Yaskawa INFORM job: N_R2_D50&56B(110_90,180).JBI

/JOB
//NAME N_R2_D50&56B(110_90,180)
//POS
///NPOS 227,227,227,10,0,0
///TOOL 0
///POSTYPE PULSE
///PULSE
C00000=22584,-91029,-87060,-7956,68824,61093
C00001=22584,-91029,-87060,-7956,68824,61093
C00002=2000,-113621,-91819,0,89172,0
C00003=-100725,-66745,-65547,-5330,101330,-31581
C00004=-137248,-37413,-60851,-11800,108062,-53976
C00005=-138411,-7940,-28391,-15115,116133,-60489
C00006=-180680,14026,-7685,-7917,112728,-80060
C00007=-186794,17026,42,-8794,108924,-82022
C00008=-187502,17265,3652,-8795,106773,-82119
C00009=-187502,17467,5395,-8744,105818,-82049
C00010=-182675,14939,3487,-14937,105773,-89393
C00011=-183307,13395,2083,-15043,105726,-89619
C00012=-186125,21667,9753,-10883,108766,-81970
C00013=-185415,19514,7722,-10739,109003,-81731
C00014=-186125,21667,9753,-10883,108766,-81970
C00015=-184476,23080,5547,-10788,112245,-81685
C00016=-135191,-11971,-32648,-15419,118418,-54869
C00017=-100725,-66745,-65547,-5330,101330,-31581
C00018=-68653,-71707,-73837,-24748,96021,-85891
C00019=-66615,-76041,-75906,-24722,95756,-75393
C00020=-80537,-30124,-13141,-12214,96831,-80465
C00021=-81172,-32496,-11329,-12285,94454,-80447
C00022=-81272,-33574,-9619,-12271,92868,-80323
C00023=-81272,-32874,-8019,-12261,92258,-80262
C00024=-81272,-33629,-9742,-12273,92916,-80327
C00025=-78377,-29561,-6671,-11651,93530,-79403
C00026=-82930,-25221,-2257,-8748,94612,-75231
C00027=-82159,-27675,-3939,-8560,94470,-74962
C00028=-82863,-25445,-2412,-8734,94601,-75208
C00029=-74565,-33759,-7503,-14334,89858,-83488
C00030=-75264,-34516,-7988,-14469,89651,-83703
C00031=-74565,-33759,-7503,-14334,89858,-83488
C00032=-74565,-35408,-11222,-14349,91256,-83650
C00033=-81291,-32137,-11094,-12310,94476,-80493
C00034=-172905,8912,9805,-17685,104206,-63243
C00035=-172925,6267,11032,-17511,102181,-62948
C00036=-173095,5120,12140,-17457,100932,-62826
C00037=-173095,5593,13541,-17414,100341,-62739
C00038=-172934,5281,11605,-17449,101360,-62831
C00039=-170941,3628,12252,-21342,95501,-69033
C00040=-171356,2541,11657,-21403,95212,-69131
C00041=-171898,950,10316,-21496,95078,-69302
C00042=-171356,2541,11657,-21403,95212,-69131
C00043=-173384,-23451,-12356,-17546,80818,-68289
C00044=-172173,-25440,-14096,-17586,81125,-67902
C00045=-171398,-26573,-14883,-17615,81198,-67636
C00046=-172724,-25294,-15625,-17531,81978,-68221
C00047=-143557,-6163,-8686,-20929,99946,-63784
C00048=-120837,-67343,-61251,1664,69818,-16688
C00049=-136948,17886,1372,-8158,95353,34817
C00050=-143935,27041,16447,-8009,90123,32767
C00051=-145422,30777,27912,-7980,84886,32590
C00052=-145422,32553,33696,-8012,82265,32756
C00053=-145422,33252,35771,-8025,81357,32815
C00054=-143676,31208,33052,-10858,81373,33518
C00055=-142910,30429,32946,-13100,80369,33952
C00056=-145422,32553,33696,-8012,82265,32756
C00057=-145422,30263,26046,-7974,85762,32534
C00058=-138335,26720,10522,-8993,93928,34380
C00059=-116233,-46119,-51802,-8224,97287,41779
C00060=-133480,-42640,-39007,-8140,89511,36383
C00061=-136265,-42532,-35298,-8104,87026,35591
C00062=-136265,-41955,-33217,-8108,86050,35653
C00063=-136265,-41609,-32030,-8111,85502,35689
C00064=-130241,-43052,-32167,-14495,84771,37934
C00065=-129806,-42953,-31605,-15984,84419,38162
C00066=-136265,-41955,-33217,-8108,86050,35653
C00067=-135498,-43523,-38278,-8113,88415,35764
C00068=-120126,-55162,-39521,-8172,84809,41259
C00069=-122393,-53466,-34860,-8212,82600,40629
C00070=-123299,-52550,-32544,-8233,81563,40387
C00071=-123299,-52047,-31285,-8241,81052,40420
C00072=-119861,-52196,-31542,-11446,81584,41751
C00073=-120901,-52203,-31545,-11457,81438,41408
C00074=-117579,-52136,-31515,-13326,82016,42591
C00075=-116541,-52768,-33293,-13289,82934,42851
C00076=-108480,-53248,-51729,-13121,95064,44368
C00077=-47420,-68885,-70906,-7741,99292,48439
C00078=-36237,-160244,-135216,-7095,93010,52660
C00079=-129093,-142421,-132565,-35762,109729,50782
C00080=-71329,-121440,-129553,-32440,109242,60016
C00081=-82746,-156345,-133581,-29501,88252,49791
C00082=-87611,-164628,-132694,-29771,81242,44951
C00083=-87611,-163220,-131273,-29779,81110,44987
C00084=-87611,-164709,-132775,-29767,81250,44951
C00085=-71886,-183234,-128665,-42620,74703,46418
C00086=-74833,-184908,-128996,-42921,72831,45887
C00087=-69878,-185821,-129175,-42644,74882,47243
C00088=-74429,-130912,-118044,-34983,110777,51627
C00089=-96642,-141369,-123481,-29522,97914,46607
C00090=-102270,-141697,-124015,-27978,95731,45009
C00091=-102270,-141154,-122872,-27952,95353,45100
C00092=-102270,-141737,-124103,-27981,95760,45001
C00093=-104565,-143039,-124460,-28044,94592,44404
C00094=-102270,-141737,-124103,-27981,95760,45001
C00095=-98711,-140115,-125335,-27931,98364,45740
C00096=-98711,-140115,-125335,-27931,98364,45740
C00097=-98939,-140108,-124921,-27921,98063,45725
C00098=-98939,-139729,-123974,-27889,97719,45808
C00099=-98939,-140167,-125070,-27927,98118,45710
C00100=-100683,-141421,-125418,-27980,97156,45273
C00101=-98939,-140167,-125070,-27927,98118,45710
C00102=-111795,-107890,-115236,-21941,123165,45716
C00103=-111980,-110192,-116037,-21807,122478,45790
C00104=-111795,-107890,-115236,-21941,123165,45716
C00105=-109061,-111903,-121767,-16718,119614,47923
C00106=-93191,-166945,-131033,-25725,96374,76077
C00107=-115036,-47760,-82622,-24757,104770,42999
C00108=-116312,-48104,-84043,-24644,105068,42493
C00109=-102840,-160852,-129487,-27293,95258,72668
C00110=-102950,-160931,-129604,-27308,95250,72628
C00111=-100000,-171791,-131669,-28056,90664,64085
C00112=-78747,-196536,-131709,-34622,83016,61742
C00113=-97788,-192520,-135527,-30708,76481,51692
C00114=-106746,-100694,-110680,-30872,101018,41696
C00115=-100997,-102592,-114676,-31446,104330,42992
C00116=-89249,-129083,-123995,-34588,91950,50732
C00117=-86172,-104791,-113024,-36662,97722,40982
C00118=-89586,-99522,-109974,-36341,97001,39840
C00119=-94829,-122476,-117865,-35334,89182,40270
C00120=-102758,-167765,-129707,-32742,64394,36090
C00121=-107366,-177085,-128987,-33295,58194,36082
C00122=-96698,-184464,-133250,-35581,61450,39784
C00123=-94800,-127534,-127780,-31715,84055,33612
C00124=-43155,-112421,-122950,-31185,87534,31974
C00125=-47420,-68885,-70906,-7741,99292,48439
C00126=-126000,-95781,-98048,7022,72166,-3406
C00127=-136814,-5298,6863,-118,87716,-82610
C00128=-137691,-48827,-35284,-2434,91122,-80550
C00129=-137775,-50491,-32454,-2438,88526,-80529
C00130=-144669,-59546,-36087,2970,81467,-83087
C00131=-137513,-49032,-30101,-2417,87837,-80428
C00132=-137980,-52740,-33271,-2456,87865,-80585
C00133=-136492,-62619,-37659,3141,80547,-80344
C00134=-130424,-52556,-33615,-1804,88372,-78049
C00135=-130538,-50934,-36491,-1816,90972,-78124
C00136=-134151,-85638,-58323,-18397,79452,-80216
C00137=-138797,-96086,-58203,-18217,70057,-80507
C00138=-132420,-53344,-33745,-21935,100560,-82879
C00139=-132280,-50606,-30920,-21871,100287,-82777
C00140=-143411,-94723,-57726,-17890,69450,-82098
C00141=-139141,-75011,-51892,-19052,86769,-83193
C00142=-144749,-26995,-11930,-14691,82144,-88756
C00143=-145691,-31856,-11979,-19284,78923,34918
C00144=-151034,-18823,4704,-13824,76424,32875
C00145=-151885,-17656,8121,-14166,75214,33243
C00146=-146071,-19738,8912,-19797,72571,35827
C00147=-147152,-20027,7322,-19728,73103,35349
C00148=-154357,-26510,2050,-14259,74004,32525
C00149=-152793,-10987,14638,-15716,82099,47051
C00150=-151339,-11562,10959,-15494,84269,47273
C00151=-146019,7566,32377,-21507,91583,49077
C00152=-147957,4386,28538,-22011,91765,48359
C00153=-147481,5615,30408,-21882,91404,48596
C00154=-144848,5152,34234,-24760,87902,50723
C00155=-159832,9049,31418,-7877,90076,62571
C00156=-198300,39103,67536,-4454,97929,51257
C00157=-197104,34479,56425,-4037,102437,51493
C00158=-197536,32116,56558,-4191,101125,51391
C00159=-198300,39103,67536,-4454,97929,51257
C00160=-197104,34479,56425,-4037,102437,51493
C00161=-145435,-6461,7890,-19316,88952,36538
C00162=-146400,-15498,9010,-17111,65695,33326
C00163=-150585,-15374,10170,-12685,65372,31387
C00164=-152770,-11869,15298,-10806,64283,30498
C00165=-148493,-14593,14125,-17227,62697,33002
C00166=-147445,-14270,15768,-17483,62104,33493
C00167=-150113,-3203,22864,-12407,64063,31649
C00168=-146055,-7115,17417,-17271,64938,33574
C00169=-149725,-15230,11944,-14152,64155,31991
C00170=-151735,-12378,15582,-12402,63542,31128
C00171=-148493,-14593,14125,-17227,62697,33002
C00172=-147444,-14270,15768,-17483,62104,33493
C00173=-151630,-3672,21747,-10124,65019,30743
C00174=-146194,-7735,16967,-17259,64868,33530
C00175=-147475,-4629,18347,-12944,66340,32408
C00176=-148206,-3042,20742,-12396,65722,32150
C00177=-144993,-5030,19536,-17422,64931,33970
C00178=-144005,-4679,21199,-17649,64331,34434
C00179=-147636,2823,25478,-11954,66212,32247
C00180=-159106,-19550,13776,8815,42964,19188
C00181=-160396,-25842,8024,9506,43156,18510
C00182=-160846,-38877,-8267,9186,46491,18652
C00183=-135242,-58896,-27541,-11024,46290,31048
C00184=-131236,-19716,-18108,-13510,71297,30401
C00185=-125742,9237,-5161,-19148,95170,30807
C00186=-133778,21116,12925,-19165,88751,28983
C00187=-139002,23165,16841,-12610,84259,27929
C00188=-139735,27050,26410,-12647,80339,28070
C00189=-131333,83852,86286,-19552,77576,31698
C00190=-130664,85028,89109,-19628,76664,32087
C00191=-140830,29311,28641,-10243,76630,19823
C00192=-140822,20487,15972,-10139,79847,19560
C00193=-137774,20952,11850,-14015,91367,38445
C00194=-140043,21612,21108,-13993,85767,38286
C00195=-131775,32332,27698,-18854,90275,38112
C00196=-132558,32274,26377,-18889,90837,37745
C00197=-141222,18370,18010,-13785,88896,43800
C00198=-140309,22876,20563,-13758,89776,44021
C00199=-138169,21721,13740,-13740,93646,44339
C00200=-130805,23103,4773,-14711,103608,44771
C00201=-116663,7219,3956,-17874,89187,41824
C00202=-120401,-109250,-97359,-24840,84473,3177
C00203=-33343,-40457,-55475,-21499,103344,-25825
C00204=-34531,-11543,-34459,-29967,106739,-58335
C00205=-34985,-14005,-32389,-29565,104365,-57871
C00206=-36737,-22261,-38534,-25905,98770,-56845
C00207=-35068,-14396,-32319,-29531,104124,-57840
C00208=-34264,-15859,-32209,-29394,103680,-57406
C00209=-37785,-26292,-41386,-25839,98165,-57100
C00210=-51408,-66161,-65218,-24804,88768,-60125
C00211=-46082,-52942,-64392,-25322,95990,-59686
C00212=-125318,-85686,-83357,-10390,89531,-85584
C00213=-142430,-46200,-62658,-6629,112309,-68083
C00214=-144446,-28774,-42147,-7166,118928,-64884
C00215=-142051,-28438,-38322,-12128,116138,-65491
C00216=-141798,-26650,-39491,-12256,117780,-65577
C00217=-132867,-37192,-45733,-18528,111034,-75329
C00218=-139736,-34425,-43384,-12199,112330,-75757
C00219=-134344,-42414,-48468,-16185,107501,-83449
C00220=-134440,-49684,-52823,-18552,102078,-90264
C00221=-130876,-45857,-53153,-18423,104940,-89409
C00222=-105687,-60080,-69740,-12786,102006,-79760
C00223=-4529,-28570,-46683,-27101,115691,-48588
C00224=2000,-113621,-91819,0,89172,0
C00225=2000,-113621,-91819,0,89172,0
C00226=2000,-113621,-91819,0,89172,0
BC00000=166445,688033,903774
BC00001=166445,688033,903774
BC00002=87189,714591,1075229
BC00003=279836,716878,248946
BC00004=347085,767945,248946
BC00005=351734,778369,248946
BC00006=397217,806013,248946
BC00007=397217,806013,248946
BC00008=397217,806013,248946
BC00009=397217,806013,248946
BC00010=397217,806013,248946
BC00011=397217,806013,248946
BC00012=397217,806013,248946
BC00013=397217,806013,248946
BC00014=397217,806013,248946
BC00015=397217,806013,248946
BC00016=347085,767945,248946
BC00017=279836,716878,248946
BC00018=74259,715122,420956
BC00019=74259,803457,420956
BC00020=74259,803457,420956
BC00021=74259,803457,420956
BC00022=74259,803457,420956
BC00023=74259,803457,420956
BC00024=74259,803457,420956
BC00025=74259,803457,420956
BC00026=74259,803457,420956
BC00027=74259,803457,420956
BC00028=74259,803457,420956
BC00029=74259,803457,420956
BC00030=74259,803457,420956
BC00031=74259,803457,420956
BC00032=74259,803457,420956
BC00033=74259,803457,420956
BC00034=168853,805006,369390
BC00035=168853,805006,369390
BC00036=168853,805006,369390
BC00037=168853,805006,369390
BC00038=168853,805006,369390
BC00039=168853,805006,369390
BC00040=168853,805006,369390
BC00041=168853,805006,369390
BC00042=168853,805006,369390
BC00043=168853,805006,369390
BC00044=168853,805006,369390
BC00045=168853,805006,369390
BC00046=168853,805006,369390
BC00047=153069,815778,383312
BC00048=89909,820992,348340
BC00049=133900,839476,347452
BC00050=133900,839476,347452
BC00051=133900,839476,347452
BC00052=133900,839476,347452
BC00053=133900,839476,347452
BC00054=133900,839476,347452
BC00055=133900,839476,347452
BC00056=133900,839476,347452
BC00057=133900,839476,347452
BC00058=133900,839476,347452
BC00059=91689,839476,305907
BC00060=91689,839476,305907
BC00061=91689,839476,305907
BC00062=91689,839476,305907
BC00063=91689,839476,305907
BC00064=91689,839476,305907
BC00065=91689,839476,305907
BC00066=91689,839476,305907
BC00067=91689,839476,305907
BC00068=65725,786338,350532
BC00069=65725,786338,350532
BC00070=65725,786338,350532
BC00071=65725,786338,350532
BC00072=65725,786338,350532
BC00073=65725,786338,350532
BC00074=65725,786338,350532
BC00075=65725,786338,350532
BC00076=65725,786338,350532
BC00077=45615,718562,524343
BC00078=45615,718562,1072524
BC00079=367621,718562,1072524
BC00080=396988,986746,1072524
BC00081=396988,986746,1072524
BC00082=396988,986746,1072524
BC00083=396988,986746,1072524
BC00084=396988,986746,1072524
BC00085=396988,986746,1072524
BC00086=396988,986746,1072524
BC00087=396988,986746,1072524
BC00088=396988,986746,1072524
BC00089=396982,986676,1072526
BC00090=396988,986746,1072524
BC00091=396988,986746,1072524
BC00092=396988,986746,1072524
BC00093=396988,986746,1072524
BC00094=396988,986746,1072524
BC00095=396988,986746,1072524
BC00096=396988,943028,1072524
BC00097=392786,943028,1061989
BC00098=392786,943028,1061989
BC00099=392786,943028,1061989
BC00100=392786,943028,1061989
BC00101=392786,943028,1061989
BC00102=392824,960696,1061989
BC00103=392824,960696,1061989
BC00104=392824,960696,1061989
BC00105=392827,960650,1061995
BC00106=397481,962635,1061991
BC00107=398174,909238,1075175
BC00108=398174,909238,1075175
BC00109=397481,962635,1061991
BC00110=397481,962635,1061991
BC00111=397481,962635,1061991
BC00112=397481,962635,1061991
BC00113=397481,962635,1061991
BC00114=397481,962635,1061991
BC00115=397481,962635,1061991
BC00116=397481,962635,1061991
BC00117=397481,962635,1061991
BC00118=397481,962635,1061991
BC00119=397481,962635,1061991
BC00120=397481,962635,1061991
BC00121=397481,962635,1061991
BC00122=397481,962635,1061991
BC00123=397481,917581,1061991
BC00124=298896,713787,1061991
BC00125=45615,718562,524343
BC00126=94279,727282,315353
BC00127=135603,815672,503004
BC00128=127958,797752,374153
BC00129=127958,797752,374153
BC00130=127958,797752,374153
BC00131=127958,797752,374153
BC00132=127958,797752,374153
BC00133=127958,797752,374153
BC00134=127958,797752,374153
BC00135=127958,797752,374153
BC00136=104823,825619,320967
BC00137=104823,825619,320967
BC00138=104823,825619,320967
BC00139=104823,825619,320967
BC00140=104823,825619,320967
BC00141=104823,825619,320967
BC00142=130544,787227,441208
BC00143=131883,785229,447466
BC00144=131883,785229,447466
BC00145=131883,785229,447466
BC00146=131883,785229,447466
BC00147=131883,785229,447466
BC00148=131883,785229,447466
BC00149=131883,785229,447466
BC00150=131883,785229,447466
BC00151=131883,785229,447466
BC00152=131883,785229,447466
BC00153=131883,785229,447466
BC00154=131883,785229,447466
BC00155=131883,785229,447466
BC00156=178294,839754,448603
BC00157=178294,839754,448603
BC00158=178294,839754,448603
BC00159=178294,839754,448603
BC00160=178294,839754,448603
BC00161=133874,781474,455608
BC00162=135864,777719,463750
BC00163=135864,777719,463750
BC00164=135864,777719,463750
BC00165=135864,777719,463750
BC00166=135864,777719,463750
BC00167=135864,777719,463750
BC00168=135864,777719,463750
BC00169=135957,805967,463073
BC00170=135957,805967,463073
BC00171=135957,805967,463073
BC00172=135957,805967,463073
BC00173=135957,805967,463072
BC00174=135957,805967,463073
BC00175=132965,820164,450481
BC00176=132965,820164,450481
BC00177=132965,820164,450481
BC00178=132965,820164,450481
BC00179=132965,820164,450481
BC00180=132965,820164,450481
BC00181=132965,820164,450481
BC00182=132965,820164,450481
BC00183=132965,820164,450481
BC00184=129716,827479,399778
BC00185=124610,838973,320111
BC00186=124537,838635,318969
BC00187=124430,838621,318501
BC00188=124430,838621,318501
BC00189=117256,837940,287867
BC00190=117256,837940,287867
BC00191=124430,838621,318501
BC00192=124430,838621,318501
BC00193=124330,838612,318094
BC00194=124330,838612,318094
BC00195=113936,839476,281332
BC00196=113936,839476,281332
BC00197=124330,838612,318094
BC00198=124330,838612,318094
BC00199=124330,838612,318094
BC00200=122155,838793,310401
BC00201=116869,821490,397669
BC00202=133980,716569,494562
BC00203=159586,725469,294802
BC00204=173113,793666,189268
BC00205=173113,793666,189268
BC00206=173113,793666,189268
BC00207=173113,793666,189268
BC00208=173113,793666,189268
BC00209=173113,793666,189268
BC00210=173113,793666,189268
BC00211=173113,793666,189268
BC00212=297390,793666,189268
BC00213=296883,794700,189268
BC00214=296884,794700,189266
BC00215=296884,794700,189266
BC00216=296884,794700,189266
BC00217=296884,794700,189266
BC00218=296884,794700,189266
BC00219=296884,794700,189266
BC00220=296884,794700,189266
BC00221=296884,794700,189266
BC00222=256017,794359,189267
BC00223=173113,793666,267263
BC00224=87189,689489,1075229
BC00225=87189,689489,1075229
BC00226=87189,689489,1075229
EC00000=10818,-11103
EC00001=10818,1079087
EC00002=798156,1112951
EC00003=798156,1112951
EC00004=798156,1112951
EC00005=798156,1112951
EC00006=798156,1112951
EC00007=798156,1112951
EC00008=798156,1112951
EC00009=798156,1112951
EC00010=798156,1112951
EC00011=798156,1112951
EC00012=798156,1112951
EC00013=798156,1112951
EC00014=798156,1112951
EC00015=798156,1112951
EC00016=798156,1112951
EC00017=798156,1112951
EC00018=798156,1112951
EC00019=798156,1112951
EC00020=798156,1112951
EC00021=798156,1112951
EC00022=798156,1112951
EC00023=798156,1112951
EC00024=798156,1112951
EC00025=798156,1112951
EC00026=798156,1112951
EC00027=798156,1112951
EC00028=798156,1112951
EC00029=798156,1112951
EC00030=798156,1112951
EC00031=798156,1112951
EC00032=798156,1112951
EC00033=798156,1112951
EC00034=798156,1112951
EC00035=798156,1112951
EC00036=798156,1112951
EC00037=798156,1112951
EC00038=798156,1112951
EC00039=798156,1112951
EC00040=798156,1112951
EC00041=798156,1112951
EC00042=798156,1112951
EC00043=798156,1112951
EC00044=798156,1112951
EC00045=798156,1112951
EC00046=798156,1112951
EC00047=798156,1112951
EC00048=798156,1112951
EC00049=798156,1112951
EC00050=798156,1112951
EC00051=798156,1112951
EC00052=798156,1112951
EC00053=798156,1112951
EC00054=798156,1112951
EC00055=798156,1112951
EC00056=798156,1112951
EC00057=798156,1112951
EC00058=798156,1112951
EC00059=798156,1112951
EC00060=798156,1112951
EC00061=798156,1112951
EC00062=798156,1112951
EC00063=798156,1112951
EC00064=798156,1112951
EC00065=798156,1112951
EC00066=798156,1112951
EC00067=798156,1112951
EC00068=798156,1112951
EC00069=798156,1112951
EC00070=798156,1112951
EC00071=798156,1112951
EC00072=798156,1112951
EC00073=798156,1112951
EC00074=798156,1112951
EC00075=798156,1112951
EC00076=798156,1112951
EC00077=798156,1112951
EC00078=798156,1112951
EC00079=798156,1112951
EC00080=798156,1112951
EC00081=798156,1112951
EC00082=798156,1112951
EC00083=798156,1112951
EC00084=798156,1112951
EC00085=798156,1112951
EC00086=798156,1112951
EC00087=798156,1112951
EC00088=798156,1112951
EC00089=798272,1112951
EC00090=798156,1112951
EC00091=798156,1112951
EC00092=798156,1112951
EC00093=798156,1112951
EC00094=798156,1112951
EC00095=798156,1112951
EC00096=798156,1112951
EC00097=798156,1112951
EC00098=798156,1112951
EC00099=798156,1112951
EC00100=798156,1112951
EC00101=798156,1112951
EC00102=798156,1112951
EC00103=798156,1112951
EC00104=798156,1112951
EC00105=798242,1112951
EC00106=798241,1112950
EC00107=975524,1112951
EC00108=975524,1112951
EC00109=798241,1112950
EC00110=798241,1112950
EC00111=798241,1112950
EC00112=798241,1112950
EC00113=798241,1112950
EC00114=798241,1112950
EC00115=798241,1112950
EC00116=798241,1112950
EC00117=798241,1112950
EC00118=798241,1112950
EC00119=798241,1112950
EC00120=798241,1112950
EC00121=798241,1112950
EC00122=798241,1112950
EC00123=798241,1112950
EC00124=798241,1112950
EC00125=798156,1112951
EC00126=798156,1112951
EC00127=798156,1112951
EC00128=798156,1112951
EC00129=798156,1112951
EC00130=798156,1112951
EC00131=798156,1112951
EC00132=798156,1112951
EC00133=798156,1112951
EC00134=798156,1112951
EC00135=798156,1112951
EC00136=798156,1112951
EC00137=798156,1112951
EC00138=798156,1112951
EC00139=798156,1112951
EC00140=798156,1112951
EC00141=798156,1112951
EC00142=798156,1112951
EC00143=798156,1112951
EC00144=798156,1112951
EC00145=798156,1112951
EC00146=798156,1112951
EC00147=798156,1112951
EC00148=798156,1112951
EC00149=798156,1112951
EC00150=798156,1112951
EC00151=798156,1112951
EC00152=798156,1112951
EC00153=798156,1112951
EC00154=798156,1112951
EC00155=798156,1112951
EC00156=798156,1112951
EC00157=798156,1112951
EC00158=798156,1112951
EC00159=798156,1112951
EC00160=798156,1112951
EC00161=798156,1112951
EC00162=798156,1112951
EC00163=798156,1112951
EC00164=798156,1112951
EC00165=798156,1112951
EC00166=798156,1112951
EC00167=798156,1112951
EC00168=798156,1112951
EC00169=798156,1112951
EC00170=798156,1112951
EC00171=798156,1112951
EC00172=798156,1112951
EC00173=798156,1112951
EC00174=798156,1112951
EC00175=798156,1112951
EC00176=798156,1112951
EC00177=798156,1112951
EC00178=798156,1112951
EC00179=798156,1112951
EC00180=798156,1112951
EC00181=798156,1112951
EC00182=798156,1112951
EC00183=798156,1112951
EC00184=798156,1112951
EC00185=798156,1112951
EC00186=798156,1112951
EC00187=798156,1112951
EC00188=798156,1112951
EC00189=798156,1112951
EC00190=798156,1112951
EC00191=798156,1112951
EC00192=798156,1112951
EC00193=798156,1112951
EC00194=798156,1112951
EC00195=798156,1112951
EC00196=798156,1112951
EC00197=798156,1112951
EC00198=798156,1112951
EC00199=798156,1112951
EC00200=798156,1112951
EC00201=798156,1112951
EC00202=798156,1112951
EC00203=798156,1112951
EC00204=798156,1112951
EC00205=798156,1112951
EC00206=798156,1112951
EC00207=798156,1112951
EC00208=798156,1112951
EC00209=798156,1112951
EC00210=798156,1112951
EC00211=798156,1112951
EC00212=798156,1112951
EC00213=798156,1112951
EC00214=798154,1112949
EC00215=798154,1112949
EC00216=798154,1112949
EC00217=798154,1112949
EC00218=798154,1112949
EC00219=798154,1112949
EC00220=798154,1112949
EC00221=798154,1112949
EC00222=798155,1112950
EC00223=798156,1112951
EC00224=798156,1112951
EC00225=12672,1112951
EC00226=0,0
///POSTYPE BASE
///RECTAN
///RCONF 0,0,0,0,0,0,0,0,0,0,0,0,0,0,0,0,0,0,0,0,0,0,0,0
P00006=0.222,-3.123,-1.508,0.0000,0.0000,0.0000
P00024=0.145,-0.552,1.326,0.0000,0.0000,0.0000
P00025=-2.003,0.006,0.728,0.0000,0.0000,0.0000
P00026=0.562,-0.002,-0.337,0.0000,0.0000,0.0000
P00027=-0.746,0.015,-9.096,0.0000,0.0000,0.0000
P00028=-2.237,-0.018,-7.702,0.0000,0.0000,0.0000
P00029=-2.156,-0.086,-4.681,0.0000,0.0000,0.0000
P00032=1.957,0.503,-7.217,0.0000,0.0000,0.0000
///RCONF 0,0,0,0,1,0,0,0,0,0,0,0,0,0,0,0,0,0,0,0,0,0,0,0
P00033=-0.123,0.612,-5.012,0.0000,0.0000,0.0000
///RCONF 0,0,0,0,0,0,0,0,0,0,0,0,0,0,0,0,0,0,0,0,0,0,0,0
P00034=-0.304,0.773,-2.693,0.0000,0.0000,0.0000
//INST
///DATE 2025/01/28 12:02
///ATTR SC,RW
///GROUP1 RB1,BS1
///GROUP2 ST1
NOP
'N_R2_D50&56B(110_90,180)
'Down
MOVJ C00000 BC00000 VJ=100.00  +MOVJ EC00000 VJ=100.00
MOVJ C00001 BC00001 VJ=100.00  +MOVJ EC00001 VJ=100.00
MOVJ C00002 BC00002 VJ=100.00  +MOVJ EC00002 VJ=100.00
MOVJ C00003 BC00003 VJ=100.00  +MOVJ EC00003 VJ=100.00
MOVJ C00004 BC00004 VJ=100.00  +MOVJ EC00004 VJ=100.00
'Path S4514
SFTOF3D
MOVJ C00005 BC00005 VJ=100.00  +MOVJ EC00005 VJ=100.00
MOVL C00006 BC00006 V=166.7  +MOVJ EC00006 VJ=100.00
SMOVL C00007 BC00007 V=100.0  +MOVJ EC00007
SMOVL C00008 BC00008 V=66.7  +MOVJ EC00008
SREFP 3 C00009 BC00009  +REFP EC00009
CALL JOB:SEARCH-R1-S13D
SET P034 P006
SFTON3D P034
SMOVL C00010 BC00010 V=100.0  +MOVJ EC00010
SREFP 3 C00011 BC00011  +REFP EC00011
CALL JOB:SEARCH-R1-S13D
SET P034 P006
SFTON3D P034
SMOVL C00012 BC00012 V=100.0  +MOVJ EC00012
SREFP 3 C00013 BC00013  +REFP EC00013
CALL JOB:SEARCH-R1-S13D
SET P034 P006
SFTON3D P034
SMOVL C00014 BC00014 V=100.0  +MOVJ EC00014
MOVL C00015 BC00015 V=400.0  +MOVJ EC00015 VJ=100.00
'EndPath S4514
MOVJ C00016 BC00016 VJ=100.00  +MOVJ EC00016 VJ=100.00
MOVJ C00017 BC00017 VJ=100.00  +MOVJ EC00017 VJ=100.00
MOVJ C00018 BC00018 VJ=100.00  +MOVJ EC00018 VJ=100.00
MOVJ C00019 BC00019 VJ=100.00  +MOVJ EC00019 VJ=100.00
'Path S4515
SFTOF3D
MOVJ C00020 BC00020 VJ=100.00  +MOVJ EC00020 VJ=100.00
MOVL C00021 BC00021 V=400.0  +MOVJ EC00021 VJ=100.00
SMOVL C00022 BC00022 V=100.0  +MOVJ EC00022
SREFP 3 C00023 BC00023  +REFP EC00023
CALL JOB:SEARCH-R1-S13D
SET P033 P006
SFTON3D P033
SMOVL C00024 BC00024 V=100.0  +MOVJ EC00024
SMOVL C00025 BC00025 V=100.0  +MOVJ EC00025
SMOVL C00026 BC00026 V=66.7  +MOVJ EC00026
SREFP 3 C00027 BC00027  +REFP EC00027
CALL JOB:SEARCH-R1-S13D
SET P033 P006
SFTON3D P033
SMOVL C00028 BC00028 V=100.0  +MOVJ EC00028
SMOVL C00029 BC00029 V=100.0  +MOVJ EC00029
SREFP 3 C00030 BC00030  +REFP EC00030
CALL JOB:SEARCH-R1-S13D
SET P033 P006
SFTON3D P033
SMOVL C00031 BC00031 V=100.0  +MOVJ EC00031
SMOVL C00032 BC00032 V=100.0  +MOVJ EC00032
MOVL C00033 BC00033 V=400.0  +MOVJ EC00033 VJ=100.00
'EndPath S4515
'Path S4516
SFTOF3D
MOVJ C00034 BC00034 VJ=100.00  +MOVJ EC00034 VJ=100.00
MOVL C00035 BC00035 V=400.0  +MOVJ EC00035 VJ=100.00
SMOVL C00036 BC00036 V=100.0  +MOVJ EC00036
SREFP 3 C00037 BC00037  +REFP EC00037
CALL JOB:SEARCH-R1-S13D
SET P032 P006
SFTON3D P032
SMOVL C00038 BC00038 V=100.0  +MOVJ EC00038
SMOVL C00039 BC00039 V=100.0  +MOVJ EC00039
SMOVL C00040 BC00040 V=66.7  +MOVJ EC00040
SREFP 3 C00041 BC00041  +REFP EC00041
CALL JOB:SEARCH-R1-S13D
SET P032 P006
SFTON3D P032
SMOVL C00042 BC00042 V=100.0  +MOVJ EC00042
SMOVL C00043 BC00043 V=100.0  +MOVJ EC00043
SMOVL C00044 BC00044 V=100.0  +MOVJ EC00044
SREFP 3 C00045 BC00045  +REFP EC00045
CALL JOB:SEARCH-R1-S13D
SET P032 P006
SFTON3D P032
SMOVL C00046 BC00046 V=100.0  +MOVJ EC00046
'EndPath S4516
MOVJ C00047 BC00047 VJ=100.00  +MOVJ EC00047 VJ=100.00
MOVJ C00048 BC00048 VJ=100.00  +MOVJ EC00048 VJ=100.00
MOVJ C00049 BC00049 VJ=40.00  +MOVJ EC00049 VJ=100.00
'Path S4519
SFTOF3D
MOVJ C00050 BC00050 VJ=40.00  +MOVJ EC00050 VJ=100.00
MOVL C00051 BC00051 V=166.7  +MOVJ EC00051 VJ=100.00
SMOVL C00052 BC00052 V=100.0  +MOVJ EC00052
SREFP 3 C00053 BC00053  +REFP EC00053
CALL JOB:SEARCH-R1-S13D
SET P029 P006
SFTON3D P029
SMOVL C00054 BC00054 V=100.0  +MOVJ EC00054
SREFP 3 C00055 BC00055  +REFP EC00055
CALL JOB:SEARCH-R1-S13D
SET P029 P006
SFTON3D P029
SMOVL C00056 BC00056 V=100.0  +MOVJ EC00056
MOVL C00057 BC00057 V=166.7  +MOVJ EC00057 VJ=100.00
MOVL C00058 BC00058 V=333.3  +MOVJ EC00058 VJ=100.00
'EndPath S4519
MOVJ C00059 BC00059 VJ=100.00  +MOVJ EC00059 VJ=100.00
'Path S4520
SFTOF3D
MOVJ C00060 BC00060 VJ=100.00  +MOVJ EC00060 VJ=100.00
MOVL C00061 BC00061 V=166.7  +MOVJ EC00061 VJ=100.00
SMOVL C00062 BC00062 V=100.0  +MOVJ EC00062
SREFP 3 C00063 BC00063  +REFP EC00063
CALL JOB:SEARCH-R1-S13D
SET P028 P006
SFTON3D P028
SMOVL C00064 BC00064 V=100.0  +MOVJ EC00064
SREFP 3 C00065 BC00065  +REFP EC00065
CALL JOB:SEARCH-R1-S13D
SET P028 P006
SFTON3D P028
SMOVL C00066 BC00066 V=100.0  +MOVJ EC00066
MOVL C00067 BC00067 V=166.7  +MOVJ EC00067 VJ=100.00
'EndPath S4520
'Path S4521
SFTOF3D
MOVJ C00068 BC00068 VJ=20.00  +MOVJ EC00068 VJ=100.00
MOVL C00069 BC00069 V=166.7  +MOVJ EC00069 VJ=100.00
SMOVL C00070 BC00070 V=100.0  +MOVJ EC00070
SREFP 3 C00071 BC00071  +REFP EC00071
CALL JOB:SEARCH-R1-S13D
SET P027 P006
SFTON3D P027
SMOVL C00072 BC00072 V=100.0  +MOVJ EC00072
SREFP 3 C00073 BC00073  +REFP EC00073
CALL JOB:SEARCH-R1-S13D
SET P027 P006
SFTON3D P027
SMOVL C00074 BC00074 V=100.0  +MOVJ EC00074
MOVL C00075 BC00075 V=166.7  +MOVJ EC00075 VJ=100.00
MOVL C00076 BC00076 V=1000.0  +MOVJ EC00076 VJ=100.00
'EndPath S4521
MOVJ C00077 BC00077 VJ=50.00  +MOVJ EC00077 VJ=100.00
'Up
MOVJ C00078 BC00078 VJ=100.00  +MOVJ EC00078 VJ=100.00
MOVJ C00079 BC00079 VJ=100.00  +MOVJ EC00079 VJ=100.00
MOVJ C00080 BC00080 VJ=100.00  +MOVJ EC00080 VJ=30.00
'Path S4522
SFTOF3D
MOVJ C00081 BC00081 VJ=100.00  +MOVJ EC00081 VJ=100.00
SMOVL C00082 BC00082 V=100.0  +MOVJ EC00082
SREFP 3 C00083 BC00083  +REFP EC00083
CALL JOB:SEARCH-R1-S13D
SET P026 P006
SFTON3D P026
SMOVL C00084 BC00084 V=100.0  +MOVJ EC00084
SMOVL C00085 BC00085 V=100.0  +MOVJ EC00085
SREFP 3 C00086 BC00086  +REFP EC00086
CALL JOB:SEARCH-R1-S13D
SET P026 P006
SFTON3D P026
SMOVL C00087 BC00087 V=100.0  +MOVJ EC00087
MOVL C00088 BC00088 V=400.0  +MOVJ EC00088 VJ=100.00
SFTOF3D
MOVL C00089 BC00089 V=400.0  +MOVJ EC00089 VJ=100.00
SMOVL C00090 BC00090 V=100.0  +MOVJ EC00090
SREFP 3 C00091 BC00091  +REFP EC00091
CALL JOB:SEARCH-R1-S13D
SET P025 P006
SFTON3D P025
SMOVL C00092 BC00092 V=100.0  +MOVJ EC00092
SREFP 3 C00093 BC00093  +REFP EC00093
CALL JOB:SEARCH-R1-S13D
SET P025 P006
SFTON3D P025
SMOVL C00094 BC00094 V=100.0  +MOVJ EC00094
MOVL C00095 BC00095 V=400.0  +MOVJ EC00095 VJ=100.00
MOVL C00096 BC00096 V=1000.0  +MOVJ EC00096 VJ=100.00
'EndPath S4523
'Path S4524
SFTOF3D
SMOVL C00097 BC00097 V=100.0  +MOVJ EC00097
SREFP 3 C00098 BC00098  +REFP EC00098
CALL JOB:SEARCH-R1-S13D
SET P024 P006
SFTON3D P024
SMOVL C00099 BC00099 V=100.0  +MOVJ EC00099
SREFP 3 C00100 BC00100  +REFP EC00100
CALL JOB:SEARCH-R1-S13D
SET P024 P006
SFTON3D P024
SMOVL C00101 BC00101 V=100.0  +MOVJ EC00101
SMOVL C00102 BC00102 V=100.0  +MOVJ EC00102
SREFP 3 C00103 BC00103  +REFP EC00103
CALL JOB:SEARCH-R1-S13D
SET P024 P006
SFTON3D P024
SMOVL C00104 BC00104 V=100.0  +MOVJ EC00104
'EndPath S4524
'Path S4525
SFTOF3D
MOVL C00105 BC00105 V=400.0  +MOVJ EC00105 VJ=100.00
SMOVL C00106 BC00106 V=100.0 PL=0  +MOVJ EC00106
SFTON3D P024
SREFP 1 C00107 BC00107  +REFP EC00107
SREFP 2 C00108 BC00108  +REFP EC00108
MACRO1 MJ#(0) ARGF9
ARCON
SMOVL C00109 BC00109 V=9.2  +MOVJ EC00109
SMOVC C00110 BC00110 V=9.2  +MOVJ EC00110
SMOVC C00111 BC00111 V=9.2  +MOVJ EC00111
ARCON
SMOVC C00112 BC00112 V=9.2  +MOVJ EC00112
SFTON3D P025
SMOVL C00113 BC00113 V=9.2  +MOVJ EC00113
SMOVL C00114 BC00114 V=9.2  +MOVJ EC00114
ARCOF
SMOVL C00115 BC00115 V=166.7  +MOVJ EC00115
SMOVL C00116 BC00116 V=333.3  +MOVJ EC00116
SFTOF3D
SMOVL C00117 BC00117 V=166.7  +MOVJ EC00117
SFTON3D P026
SMOVL C00118 BC00118 V=100.0 PL=0  +MOVJ EC00118
MACRO1 MJ#(0) ARGF14
ARCON
SMOVL C00119 BC00119 V=7.5  +MOVJ EC00119
SMOVL C00120 BC00120 V=7.5  +MOVJ EC00120
SMOVL C00121 BC00121 V=8.3  +MOVJ EC00121
ARCOF
SMOVL C00122 BC00122 V=166.7  +MOVJ EC00122
SMOVL C00123 BC00123 V=1000.0  +MOVJ EC00123
MOVJ C00124 BC00124 VJ=100.00  +MOVJ EC00124 VJ=100.00
'EndPath W4531
'Down
MOVJ C00125 BC00125 VJ=100.00  +MOVJ EC00125 VJ=100.00
MOVJ C00126 BC00126 VJ=100.00  +MOVJ EC00126 VJ=100.00
SFTOF3D
'EndPath W4533
MOVJ C00127 BC00127 VJ=100.00  +MOVJ EC00127 VJ=100.00
'Path W4534
SFTOF3D
SFTON3D P033
MOVJ C00128 BC00128 VJ=100.00  +MOVJ EC00128 VJ=100.00
SMOVL C00129 BC00129 V=400.0  +MOVJ EC00129
SMOVL C00130 BC00130 V=100.0 PL=0  +MOVJ EC00130
SREFP 1 C00131 BC00131  +REFP EC00131
SREFP 2 C00132 BC00132  +REFP EC00132
MACRO1 MJ#(0) ARGF14
ARCON
SMOVL C00133 BC00133 V=10.0  +MOVJ EC00133
ARCOF
SMOVL C00134 BC00134 V=400.0  +MOVJ EC00134
SMOVL C00135 BC00135 V=1000.0  +MOVJ EC00135
SFTOF3D
'EndPath W4534
'Path W4535
SFTOF3D
SFTON3D P032
MOVJ C00136 BC00136 VJ=100.00  +MOVJ EC00136 VJ=100.00
SMOVL C00137 BC00137 V=100.0 PL=0  +MOVJ EC00137
SREFP 1 C00138 BC00138  +REFP EC00138
SREFP 2 C00139 BC00139  +REFP EC00139
MACRO1 MJ#(0) ARGF14
ARCON
SMOVL C00140 BC00140 V=11.7  +MOVJ EC00140
ARCOF
SMOVL C00141 BC00141 V=400.0  +MOVJ EC00141
MOVJ C00142 BC00142 VJ=15.00  +MOVJ EC00142 VJ=15.00
SFTOF3D
SFTON3D P027
MOVJ C00143 BC00143 VJ=100.00  +MOVJ EC00143 VJ=100.00
SMOVL C00144 BC00144 V=133.3  +MOVJ EC00144
SMOVL C00145 BC00145 V=83.3 PL=0  +MOVJ EC00145
SREFP 1 C00146 BC00146  +REFP EC00146
SREFP 2 C00147 BC00147  +REFP EC00147
MACRO1 MJ#(0) ARGF14
ARCON
SMOVL C00148 BC00148 V=10.0  +MOVJ EC00148
SMOVL C00149 BC00149 V=10.0  +MOVJ EC00149
ARCOF
SMOVL C00150 BC00150 V=400.0  +MOVJ EC00150
SFTOF3D
SFTON3D P032
SMOVL C00151 BC00151 V=166.7  +MOVJ EC00151
SMOVL C00152 BC00152 V=166.7 PL=0  +MOVJ EC00152
ARCON
SMOVL C00153 BC00153 V=12.5  +MOVJ EC00153
SMOVL C00154 BC00154 V=12.5  +MOVJ EC00154
SMOVL C00155 BC00155 V=12.5  +MOVJ EC00155
SMOVL C00156 BC00156 V=14.2  +MOVJ EC00156
ARCOF
SMOVL C00157 BC00157 V=166.7  +MOVJ EC00157
SMOVL C00158 BC00158 V=166.7 PL=0  +MOVJ EC00158
ARCON
SMOVL C00159 BC00159 V=14.2  +MOVJ EC00159
ARCOF
SMOVL C00160 BC00160 V=166.7  +MOVJ EC00160
SFTOF3D
'EndPath W4537
MOVJ C00161 BC00161 VJ=100.00  +MOVJ EC00161 VJ=100.00
'Path W4538
SFTOF3D
SFTON3D P027
MOVJ C00162 BC00162 VJ=100.00  +MOVJ EC00162 VJ=100.00
SMOVL C00163 BC00163 V=166.7  +MOVJ EC00163
SMOVL C00164 BC00164 V=83.3 PL=0  +MOVJ EC00164
SREFP 1 C00165 BC00165  +REFP EC00165
SREFP 2 C00166 BC00166  +REFP EC00166
MACRO1 MJ#(0) ARGF0
ARCON
SMOVL C00167 BC00167 V=10.0  +MOVJ EC00167
ARCOF
SMOVL C00168 BC00168 V=166.7  +MOVJ EC00168
SFTOF3D
'EndPath W4538
'Path W4539
SFTOF3D
SFTON3D P028
SMOVL C00169 BC00169 V=166.7  +MOVJ EC00169
SMOVL C00170 BC00170 V=83.3 PL=0  +MOVJ EC00170
SREFP 1 C00171 BC00171  +REFP EC00171
SREFP 2 C00172 BC00172  +REFP EC00172
MACRO1 MJ#(0) ARGF14
ARCON
SMOVL C00173 BC00173 V=10.0  +MOVJ EC00173
ARCOF
SMOVL C00174 BC00174 V=166.7  +MOVJ EC00174
SFTOF3D
SFTON3D P028
SMOVL C00175 BC00175 V=166.7  +MOVJ EC00175
SMOVL C00176 BC00176 V=150.0 PL=0  +MOVJ EC00176
SREFP 1 C00177 BC00177  +REFP EC00177
SREFP 2 C00178 BC00178  +REFP EC00178
MACRO1 MJ#(0) ARGF14
ARCON
SMOVL C00179 BC00179 V=10.0  +MOVJ EC00179
SMOVL C00180 BC00180 V=10.0  +MOVJ EC00180
ARCOF
SMOVL C00181 BC00181 V=83.3  +MOVJ EC00181
SMOVL C00182 BC00182 V=250.0  +MOVJ EC00182
SFTOF3D
'EndPath W4540
MOVJ C00183 BC00183 VJ=100.00  +MOVJ EC00183 VJ=100.00
MOVJ C00184 BC00184 VJ=100.00  +MOVJ EC00184 VJ=100.00
MOVJ C00185 BC00185 VJ=100.00  +MOVJ EC00185 VJ=100.00
'Path W4541
SFTOF3D
SFTON3D P029
MOVJ C00186 BC00186 VJ=100.00  +MOVJ EC00186 VJ=100.00
SMOVL C00187 BC00187 V=166.7  +MOVJ EC00187
SMOVL C00188 BC00188 V=100.0 PL=0  +MOVJ EC00188
SREFP 1 C00189 BC00189  +REFP EC00189
SREFP 2 C00190 BC00190  +REFP EC00190
MACRO1 MJ#(0) ARGF14
ARCON
SMOVL C00191 BC00191 V=10.0  +MOVJ EC00191
ARCOF
SMOVL C00192 BC00192 V=166.7  +MOVJ EC00192
SMOVL C00193 BC00193 V=333.3  +MOVJ EC00193
SFTOF3D
'EndPath W4541
'Path W4542
SFTOF3D
SFTON3D P029
SMOVL C00194 BC00194 V=150.0 PL=0  +MOVJ EC00194
SREFP 1 C00195 BC00195  +REFP EC00195
SREFP 2 C00196 BC00196  +REFP EC00196
MACRO1 MJ#(0) ARGF14
ARCON
SMOVL C00197 BC00197 V=10.0  +MOVJ EC00197
ARCOF
SMOVL C00198 BC00198 V=133.3  +MOVJ EC00198
SMOVL C00199 BC00199 V=250.0  +MOVJ EC00199
SFTOF3D
'EndPath W4542
MOVJ C00200 BC00200 VJ=15.00  +MOVJ EC00200 VJ=100.00
MOVJ C00201 BC00201 VJ=100.00  +MOVJ EC00201 VJ=100.00
MOVJ C00202 BC00202 VJ=100.00  +MOVJ EC00202 VJ=100.00
MOVJ C00203 BC00203 VJ=100.00  +MOVJ EC00203 VJ=100.00
'Path W4543
SFTOF3D
SFTON3D P034
MOVJ C00204 BC00204 VJ=100.00  +MOVJ EC00204 VJ=100.00
SMOVL C00205 BC00205 V=400.0  +MOVJ EC00205
SMOVL C00206 BC00206 V=150.0 PL=0  +MOVJ EC00206
SREFP 1 C00207 BC00207  +REFP EC00207
SREFP 2 C00208 BC00208  +REFP EC00208
MACRO1 MJ#(0) ARGF14
ARCON
SMOVL C00209 BC00209 V=11.7  +MOVJ EC00209
SMOVL C00210 BC00210 V=11.7  +MOVJ EC00210
ARCOF
SMOVL C00211 BC00211 V=250.0  +MOVJ EC00211
MOVJ C00212 BC00212 VJ=15.00  +MOVJ EC00212 VJ=15.00
MOVJ C00213 BC00213 VJ=10.00  +MOVJ EC00213 VJ=15.00
SMOVL C00214 BC00214 V=83.3  +MOVJ EC00214
ARCON
SMOVL C00215 BC00215 V=10.0  +MOVJ EC00215
ARCOF
SMOVL C00216 BC00216 V=25.0  +MOVJ EC00216
SMOVL C00217 BC00217 V=25.0  +MOVJ EC00217
SMOVL C00218 BC00218 V=25.0  +MOVJ EC00218
ARCON
SMOVL C00219 BC00219 V=10.0  +MOVJ EC00219
SMOVL C00220 BC00220 V=10.0  +MOVJ EC00220
ARCOF
SMOVL C00221 BC00221 V=100.0  +MOVJ EC00221
SMOVL C00222 BC00222 V=166.7  +MOVJ EC00222
SFTOF3D
'EndPath W4543
MOVJ C00223 BC00223 VJ=100.00  +MOVJ EC00223 VJ=100.00
MOVJ C00224 BC00224 VJ=100.00  +MOVJ EC00224 VJ=100.00
MOVJ C00225 BC00225 VJ=100.00  +MOVJ EC00225 VJ=100.00
MOVJ C00226 BC00226 VJ=100.00  +MOVJ EC00226 VJ=100.00
END
